FUNCTION_BLOCK DefaultParameters
VAR_INPUT
	Pressure: ControllerParameters := ( P := 0.02, I := T#2M );
	Flow: ControllerParameters := ( P := 0.02, I := T#2M );
	SlaveFlow: ControllerParameters := ( P := 0.02, I := T#2M );
	Const: ControllerParameters := ( P := 0.02, I := T#2M );
END_VAR
VAR_OUTPUT
END_VAR
VAR
END_VAR

END_FUNCTION_BLOCK

(* stored: Version 1.1.0.1, ProductVersion 3.1.4024.6
   POU DefaultParameters: Id {4975ba0a-01f7-4cdb-a2ac-96db5e0f2562}, SpecialFunc None *)
